# EPICS autosave request: iocBoot/iocNSLS2_EM/auto_settings.req
file "NSLS2_EM_settings.req",          P=$(P), R=$(R)
file "quadEM_settings.req",            P=$(P), R=$(R)
file "quadEM_Plugin_settings.req",     P=$(P), R=$(R)
